INTERFACE I_Button

PROPERTY IsPressed : BOOL
GET
END_GET
END_PROPERTY

PROPERTY IsReleased : BOOL
GET
END_GET
END_PROPERTY

PROPERTY RisingTrigger : BOOL
GET
END_GET
END_PROPERTY

END_INTERFACE

(* stored: Version 1.1.0.1
   Itf I_Button: Id {d489b1a5-a2f1-4e4c-bd4f-d64b53deabd3}
   Property IsPressed: Id {c5fef8e3-b7de-450e-8669-299152d81b7d}
   Get Get: Id {473dc3c8-bcb4-4776-abd5-54dccfd466fb}
   Property IsReleased: Id {8e1dc4a3-b2bb-457b-8eb1-dfcc1b45ab27}
   Get Get: Id {3d0f138f-fc04-4888-b61d-d086135a7138}
   Property RisingTrigger: Id {9710214a-b738-4d97-98ac-ff35a60f2368}
   Get Get: Id {d3a539f2-4c5f-48c3-a2a7-c8c4d8425de2} *)
